FUNCTION_BLOCK INTERNAL FB_State2 EXTENDS FB_State
VAR_INPUT
END_VAR
VAR_OUTPUT
END_VAR
VAR
END_VAR

END_FUNCTION_BLOCK

(* stored: Version 1.1.0.1, ProductVersion 3.1.4024.12
   POU FB_State2: Id {664c458a-2b42-067d-2de7-1ca31cb909c6}, SpecialFunc None *)
